// TIA Portal project "TEST TCP" (V16)

(* hardware
DEVICE "S7-1200 station_1"  S7-1200 Station
   slot 0: "Rack_0"  S7-1200 Rack  Rack  V1.0
   slot 1: "PLC_1"  CPU 1214C DC/DC/DC  6ES7 214-1AG40-0XB0  V4.2
   slot 2: "AI 4x13BIT/AQ 2x14BIT_1"  6ES7 234-4HE32-0XB0  V2.1
*)

// ===== PLC "PLC_1"  CPU 1214C DC/DC/DC =====

VAR_GLOBAL   // PLC tag table "Default tag table"
   "SET" AT %MW0 : Int;
END_VAR

DATA_BLOCK "DATA TCP"   // DB1
{ S7_Optimized_Access := 'FALSE' }
VERSION : 0.1
   VAR
      DATA : Array[0..9] of Int;
   END_VAR
BEGIN
END_DATA_BLOCK

DATA_BLOCK "MB Config"   // DB3
{ S7_Optimized_Access := 'FALSE' }
VERSION : 0.1
   VAR
      CONNECT : TCON_IP_v4;
   END_VAR
BEGIN
   CONNECT.InterfaceId := 64;
   CONNECT.ID := 1;
   CONNECT.ConnectionType := 11;
   CONNECT.RemoteAddress.ADDR[1] := 192;
   CONNECT.RemoteAddress.ADDR[2] := 168;
   CONNECT.RemoteAddress.ADDR[3] := 0;
   CONNECT.RemoteAddress.ADDR[4] := 100;
   CONNECT.LocalPort := 502;
END_DATA_BLOCK

ORGANIZATION_BLOCK "Main"   // OB1, LAD, ProgramCycle
TITLE = "Main Program Sweep (Cycle)"
{ S7_Optimized_Access := 'TRUE' }
VERSION : 0.1
   VAR_INPUT
      Initial_Call : Bool;   // Initial call of this OB
      Remanence : Bool;   // =True, if remanent data are available
   END_VAR
BEGIN

REGION Network 1
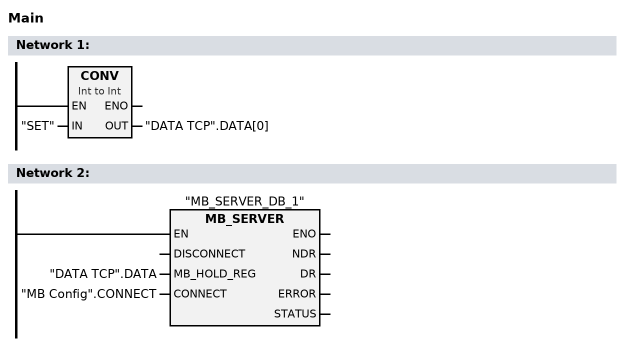
   RUNG wire#powerrail
      { S7_Templates := "[SrcType := Int, DestType := Int]" } Convert(in := "SET", out => "DATA TCP".DATA[0])
   END_RUNG
   // the same network as SCL:
   "DATA TCP".DATA[0] := INT_TO_INT("SET");
END_REGION

REGION Network 2
   "MB_SERVER_DB_1"(MB_HOLD_REG := "DATA TCP".DATA, CONNECT := "MB Config".CONNECT);   // MB_SERVER
END_REGION
END_ORGANIZATION_BLOCK